Fanuc KAREL source: kf00070.KL

-- PROVISIONAL review KL for V940-1; original PC SHA256 0d807363afbe2b11ca90be47c8317a51688fc536bf067703e6b15e29c9313ad0
-- Incomplete behavior may be omitted. Consult companion uncertainty JSON. Do not deploy.
PROGRAM KF00070
%NOLOCKGROUP
VAR
  I : INTEGER
  J : INTEGER
  X : REAL
  Y : REAL
  B : BOOLEAN
  C : BOOLEAN
  TXT : STRING[80]
  TXT2 : STRING[80]
  STATUS : INTEGER
-- UNRESOLVED_DECL AI type=002010
-- UNRESOLVED_DECL BI type=002010
-- UNRESOLVED_DECL P type=000102
-- UNRESOLVED_DECL JP type=000199
-- UNRESOLVED_DECL PF type=000101
-- UNRESOLVED_DECL V1 type=000013
-- UNRESOLVED_DECL V2 type=000013
BEGIN
  -- V9_ZERO_TABLE_METADATA_HINT layout=0001; no indexed target words; source/name/runtime held
  -- UNRESOLVED_PC offsets 5-15; opcodes 3F,75
  -- UNRESOLVED_PC offsets 20-29; opcodes 3F,75
  -- UNRESOLVED_PC offsets 34-45; opcodes 2E,23
  -- UNRESOLVED_PC offsets 50-61; opcodes 2E,23
  -- UNRESOLVED_PC offsets 66-79; opcodes 22,1D,23
  -- UNRESOLVED_PC offsets 84-88; opcodes 7F
END KF00070
